// TIA Portal V21 export
ORGANIZATION_BLOCK "Main"   // OB1, LAD, ProgramCycle
TITLE = Main loop
{ S7_Optimized_Access := 'TRUE' }
// stored: SetENOAutomatically false
   VAR_INPUT
      Initial_Call : Bool;
      Remanence : Bool;
   END_VAR
BEGIN

REGION Network 1: Konnektierungsbaustein für PLC-Lab
   // #Deutsch (#English below)
   // Im Netzwerk 1 wird der Konnektierungsbaustein für PLC-Lab aufgerufen.
   // Dieser Aufruf darf nicht entfernt werden!
   // 
   // #English
   // The connection block for PLC-Lab is called up in network 1.
   // This call must not be removed!
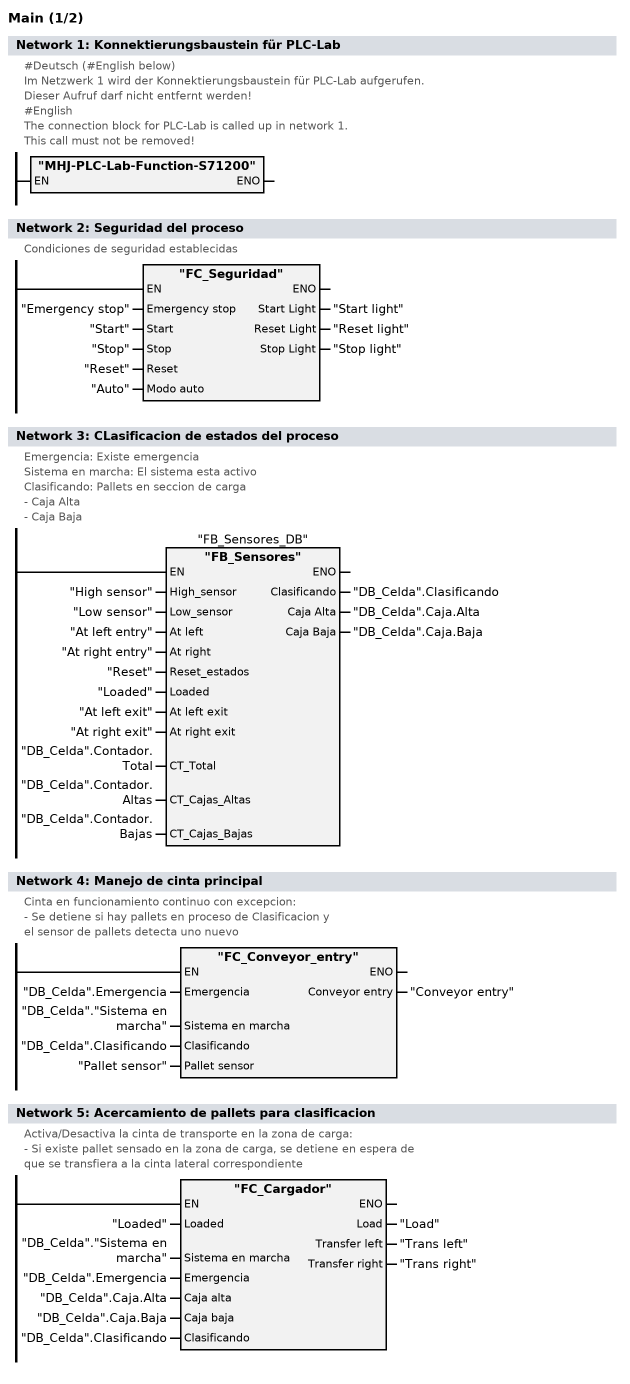
   RUNG wire#powerrail
      "MHJ-PLC-Lab-Function-S71200"()
   END_RUNG
   // the same network as SCL:
   "MHJ-PLC-Lab-Function-S71200"();
END_REGION

REGION Network 2: Seguridad del proceso
   // Condiciones de seguridad establecidas
   RUNG wire#powerrail
      "FC_Seguridad"("Emergency stop" := "Emergency stop", Start := "Start", Stop := "Stop", Reset := "Reset", "Modo auto" := "Auto", "Start Light" => "Start light", "Reset Light" => "Reset light", "Stop Light" => "Stop light")
   END_RUNG
   // the same network as SCL:
   "FC_Seguridad"("Emergency stop" := "Emergency stop",
                  Start := "Start",
                  Stop := "Stop",
                  Reset := "Reset",
                  "Modo auto" := "Auto",
                  "Start Light" => "Start light",
                  "Reset Light" => "Reset light",
                  "Stop Light" => "Stop light");
END_REGION

REGION Network 3: CLasificacion de estados del proceso
   // Emergencia: Existe emergencia
   // Sistema en marcha: El sistema esta activo
   // Clasificando: Pallets en seccion de carga
   // - Caja Alta
   // - Caja Baja
   RUNG wire#powerrail
      "FB_Sensores_DB"(High_sensor := "High sensor", Low_sensor := "Low sensor", "At left" := "At left entry", "At right" := "At right entry", Reset_estados := "Reset", Loaded := "Loaded", "At left exit" := "At left exit", "At right exit" := "At right exit", CT_Total := "DB_Celda".Contador.Total, CT_Cajas_Altas := "DB_Celda".Contador.Altas, CT_Cajas_Bajas := "DB_Celda".Contador.Bajas, Clasificando => "DB_Celda".Clasificando, "Caja Alta" => "DB_Celda".Caja.Alta, "Caja Baja" => "DB_Celda".Caja.Baja)
   END_RUNG
   // the same network as SCL:
   "FB_Sensores_DB"(High_sensor := "High sensor",   // "FB_Sensores"
                    Low_sensor := "Low sensor",
                    "At left" := "At left entry",
                    "At right" := "At right entry",
                    Reset_estados := "Reset",
                    Loaded := "Loaded",
                    "At left exit" := "At left exit",
                    "At right exit" := "At right exit",
                    CT_Total := "DB_Celda".Contador.Total,
                    CT_Cajas_Altas := "DB_Celda".Contador.Altas,
                    CT_Cajas_Bajas := "DB_Celda".Contador.Bajas,
                    Clasificando => "DB_Celda".Clasificando,
                    "Caja Alta" => "DB_Celda".Caja.Alta,
                    "Caja Baja" => "DB_Celda".Caja.Baja);
END_REGION

REGION Network 4: Manejo de cinta principal
   // Cinta en funcionamiento continuo con excepcion:
   // - Se detiene si hay pallets en proceso de Clasificacion y 
   //   el sensor de pallets detecta uno nuevo
   RUNG wire#powerrail
      "FC_Conveyor_entry"(Emergencia := "DB_Celda".Emergencia, "Sistema en marcha" := "DB_Celda"."Sistema en marcha", Clasificando := "DB_Celda".Clasificando, "Pallet sensor" := "Pallet sensor", "Conveyor entry" => "Conveyor entry")
   END_RUNG
   // the same network as SCL:
   "FC_Conveyor_entry"(Emergencia := "DB_Celda".Emergencia,
                       "Sistema en marcha" := "DB_Celda"."Sistema en marcha",
                       Clasificando := "DB_Celda".Clasificando,
                       "Pallet sensor" := "Pallet sensor",
                       "Conveyor entry" => "Conveyor entry");
END_REGION

REGION Network 5: Acercamiento de pallets para clasificacion
   // Activa/Desactiva la cinta de transporte en la zona de carga:
   // - Si existe pallet sensado en la zona de carga, se detiene en espera de
   //   que se transfiera a la cinta lateral correspondiente
   RUNG wire#powerrail
      "FC_Cargador"(Loaded := "Loaded", "Sistema en marcha" := "DB_Celda"."Sistema en marcha", Emergencia := "DB_Celda".Emergencia, "Caja alta" := "DB_Celda".Caja.Alta, "Caja baja" := "DB_Celda".Caja.Baja, Clasificando := "DB_Celda".Clasificando, Load => "Load", "Transfer left" => "Trans left", "Transfer right" => "Trans right")
   END_RUNG
   // the same network as SCL:
   "FC_Cargador"(Loaded := "Loaded",
                 "Sistema en marcha" := "DB_Celda"."Sistema en marcha",
                 Emergencia := "DB_Celda".Emergencia,
                 "Caja alta" := "DB_Celda".Caja.Alta,
                 "Caja baja" := "DB_Celda".Caja.Baja,
                 Clasificando := "DB_Celda".Clasificando,
                 Load => "Load",
                 "Transfer left" => "Trans left",
                 "Transfer right" => "Trans right");
END_REGION

REGION Network 6: Manejo de Cintas Laterales
   // Siempre activas si el sistema esta en marcha
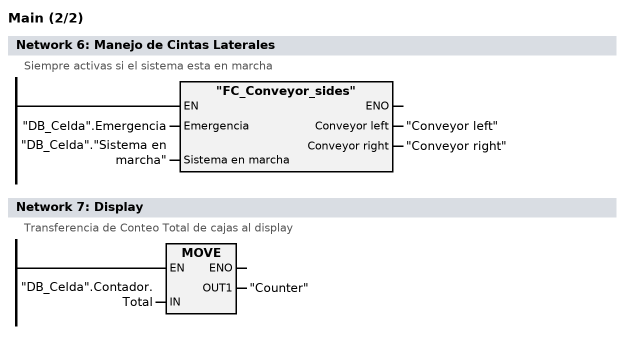
   RUNG wire#powerrail
      "FC_Conveyor_sides"(Emergencia := "DB_Celda".Emergencia, "Sistema en marcha" := "DB_Celda"."Sistema en marcha", "Conveyor left" => "Conveyor left", "Conveyor right" => "Conveyor right")
   END_RUNG
   // the same network as SCL:
   "FC_Conveyor_sides"(Emergencia := "DB_Celda".Emergencia,
                       "Sistema en marcha" := "DB_Celda"."Sistema en marcha",
                       "Conveyor left" => "Conveyor left",
                       "Conveyor right" => "Conveyor right");
END_REGION

REGION Network 7: Display
   // Transferencia de Conteo Total de cajas al display
   RUNG wire#powerrail
      Move(in := "DB_Celda".Contador.Total, out1 => "Counter")
   END_RUNG
   // the same network as SCL:
   "Counter" := "DB_Celda".Contador.Total;
END_REGION
END_ORGANIZATION_BLOCK
